FUNCTION_BLOCK FB_AxisPTP EXTENDS FB_Axis
VAR_INPUT
END_VAR
VAR_OUTPUT
END_VAR
VAR
	// ================== Axis function block =================
	fbMcMove	: MC_MoveVelocity;
	fbMcHalt	: MC_Halt;
	fbMcMovePos	: MC_MoveAbsolute;
	
	// ================== Trigger ==============================
	rTrigHalt		: R_TRIG;
	rTrigMove		: R_TRIG;
	rTrigMovePos	: R_TRIG;
END_VAR

METHOD PUBLIC  M_Halt : BOOL
VAR_INPUT
	bExecute	:	BOOL;
END_VAR
IF NOT bExecute THEN
	bHaltDone := FALSE;
ELSE
	fbMcMove(	Axis	:= Axis,
				Execute := FALSE);
END_IF

rTrigHalt(CLK := bExecute);

IF rTrigHalt.Q THEN
	fbMcHalt(	Axis	:= Axis,
				Execute	:= TRUE);
ELSE
	fbMcHalt(	Axis	:= Axis);
END_IF

IF fbMcHalt.Done OR fbMcHalt.Error OR fbMcHalt.CommandAborted THEN
	bError		:= fbMcHalt.Error;
	nErrorID	:= fbMcHalt.ErrorID;
	bHaltDone	:= fbMcHalt.Done;
	
	fbMcHalt(	Axis	:= Axis,
				Execute	:= FALSE);
END_IF
END_METHOD

METHOD M_MoveFw : BOOL
VAR_INPUT
	bExecute	: BOOL;
END_VAR
IF _fVelocity <= 0 THEN
	bExecute := FALSE;
END_IF

IF bExecute THEN
	fbMcMovePos(Axis := Axis, Execute := FALSE);
ELSE
	;
END_IF

rTrigMove(CLK := bExecute);

IF rTrigMove.Q THEN
	fbMcMove(	Axis		:= Axis,
				Execute		:= TRUE,
				Velocity	:= _fVelocity,
				Direction	:= MC_Positive_Direction);
END_IF

// Error, Command aborted
IF fbMcMove.Error OR fbMcMove.CommandAborted THEN
	bError		:= fbMcMove.Error;
	nErrorID	:= fbMcMove.ErrorID;
	
	fbMcMove(	Axis	:= Axis,
				Execute	:= FALSE);
END_IF
END_METHOD

METHOD PUBLIC M_MovePos : BOOL
VAR_INPUT
	bExecute	: BOOL;
END_VAR
IF _fVelocity <= 0 THEN
	bExecute := FALSE;
END_IF

IF bExecute THEN
	fbMcMove(Axis := Axis, Execute := FALSE);
ELSE
	bMovePosDone := FALSE;
END_IF

rTrigMovePos(CLK := bExecute);

IF rTrigMovePos.Q THEN
	fbMcMovePos(	Axis		:= Axis,
					Execute		:= TRUE,
					Position	:= _fPosition,
					Velocity	:= _fVelocity);
ELSE
	fbMcMovePos(	Axis		:= Axis);
END_IF
		
IF fbMcMovePos.Done OR fbMcMovePos.CommandAborted OR fbMcMovePos.Error THEN
	bMovePosDone	:= fbMcMovePos.Done;
	bError			:= fbMcMovePos.Error;
	nErrorID		:= fbMcMovePos.ErrorID;
	
	fbMcMovePos(Axis := Axis, Execute := FALSE);
END_IF
END_METHOD

METHOD M_Reset : BOOL
VAR_INPUT
	bExecute	: BOOL;
END_VAR
SUPER^.M_Reset(bExecute := bExecute);

IF bExecute THEN
	fbMcMove(	Axis := Axis,
			Execute := FALSE);

	fbMcHalt(	Axis := Axis,
				Execute := FALSE);
END_IF
END_METHOD

END_FUNCTION_BLOCK

(* stored: Version 1.1.0.1, ProductVersion 3.1.4024.6
   POU FB_AxisPTP: Id {a6a38ca3-1810-406b-b014-1f56a4f6209e}, SpecialFunc None
   Method M_Halt: Id {32557a7c-dcf1-41ea-8258-b3e71d43fdfa}
   Method M_MoveFw: Id {82f380d0-e82a-4411-a8f9-af52a89203e4}
   Method M_MovePos: Id {a7016dbb-48c9-47d3-b0e4-8214228031fb}
   Method M_Reset: Id {7f47d796-b985-4399-855f-b4844c2f5ace} *)
